FUNCTION_BLOCK FB_AxisControl EXTENDS FB_McAxis
VAR
  _eCheck                   : E_CHECK_STATE;  // pointer check

  _eAxisCycle,                                // cyclic AXIS_REF() and MC_Power check
  _eInit                    : E_PROGRESS;     // axis startup and init, get encoder type, get axis name

  _nAxisIndex               : UINT;           // know thyself
  _rTargetWindow            : LREAL := 0.1;   // TODO: get that from NC

  _stCtrl                   : POINTER TO ARRAY[1..PLC_CONSTANT.MAX_AXIS] OF ST_AXIS_CTRL;
  _stState                  : POINTER TO ARRAY[1..PLC_CONSTANT.MAX_AXIS] OF ST_AXIS_STATE;

  _Info                     : POINTER TO ARRAY[1..PLC_CONSTANT.MAX_AXIS] OF ST_AXIS_INFO;    // axis state and position data to read from
  _Data                     : POINTER TO ARRAY[1..PLC_CONSTANT.MAX_AXIS] OF ST_MOVE_DATA;    // structure for cyclic interface

  _NcParameter              : POINTER TO ARRAY[1..PLC_CONSTANT.MAX_AXIS] OF ST_NC_PARAMETER; // R/W struct for a single parameter
  _HomeParameter            : POINTER TO ARRAY[1..PLC_CONSTANT.MAX_AXIS] OF ST_HOMING;       // homing parameter for each axis

  _GearInParameter          : POINTER TO ARRAY[1..PLC_CONSTANT.MAX_AXIS] OF ST_GEAR_IN;
  _GearMultiMasterParameter : POINTER TO ARRAY[1..PLC_CONSTANT.MAX_AXIS] OF ST_GEAR_IN;

  _MotionOptions            : POINTER TO ARRAY[1..PLC_CONSTANT.MAX_AXIS] OF ST_MOTION_OPTIONS;


  _eCtrl,
  _eCtrlOld                 : E_AXIS_CTRL;

  _eCtrlParameterNr         : Tc2_MC2.MC_AxisParameter;

  _rParameterReadValue,
  _rParameterWrtValue       : LREAL;

  _eResult,
  _eResultOld               : E_PROGRESS;
  _eState                   : E_AXIS_STATE;

  // calibration options with limit switches and simulation
  _bCalibrationCam                : BOOL;

  _bLimitMin,
  _bLimitMax,
  _bCalibrationInput     AT %I*   : BOOL;
END_VAR

IF NOT Check() THEN RETURN; END_IF
//-----------------------------------------------------------------------------
// check _HomeParameter for calibration input options
//-----------------------------------------------------------------------------
_bCalibrationCam                    := GetCalibrationCam();
CalibrationCam                      := ADR(_bCalibrationCam);
//-----------------------------------------------------------------------------
//-----------------------------------------------------------------------------
Override                            := _Data^[_nAxisIndex].rOverride;


//-----------------------------------------------------------------------------
//-----------------------------------------------------------------------------
// cyclic call to MC_Power and AXIS_REF()
//-----------------------------------------------------------------------------
_eAxisCycle                         := Cycle();
//-----------------------------------------------------------------------------
//-----------------------------------------------------------------------------
// get command from outside world
//-----------------------------------------------------------------------------
_eCtrl                              := _stCtrl^[_nAxisIndex].eCtrl;

IF (_eCtrl <> _eCtrlOld)
THEN
  _eState                           := Cmd(_eCtrl);
  _eCtrlOld                         := _eCtrl;

  LogControl();

  _stState^[_nAxisIndex].eState     := _eState + TO_UINT(E_PROGRESS.BUSY);
END_IF
//-----------------------------------------------------------------------------
//-----------------------------------------------------------------------------
CASE _eState
OF
  E_AXIS_STATE.AXIS_INIT:
    //-------------------------------------------------------------------------
    // axis always requires one init from outside world at startup
    // _eInit has to be valid for other commands to be accepted in Cmd(_eCtrl)
    _eInit := _eResult              := AxisInit(TRUE);
    //-------------------------------------------------------------------------

  E_AXIS_STATE.AXIS_DISABLE:
    _eResult                        := AxisDisable(TRUE);

  E_AXIS_STATE.AXIS_ENABLE:
    _eResult                        := AxisEnable(TRUE);

  E_AXIS_STATE.AXIS_IDLE:
    _eResult                        := Idle(TRUE);

  E_AXIS_STATE.AXIS_HOME:
    _eResult                        := AxisHome(TRUE);

  E_AXIS_STATE.AXIS_MOVE_POS:
    _eResult                        := MovePosition(TRUE, _Data^[_nAxisIndex]);

  E_AXIS_STATE.AXIS_MOVE_VELO:
    _eResult                        := MoveVelocity(TRUE, _Data^[_nAxisIndex]);

  E_AXIS_STATE.AXIS_RESET:
    _eResult                        := AxisReset(TRUE);

  E_AXIS_STATE.AXIS_HALT:
    _eResult                        := AxisHalt(TRUE, _Data^[_nAxisIndex]);

  E_AXIS_STATE.AXIS_STOP:
    _eResult                        := AxisStop(TRUE, _Data^[_nAxisIndex]);

  E_AXIS_STATE.AXIS_MOVE_BUFFER:
    _eResult                        := MoveBufferPos(TRUE, _Data^[_nAxisIndex]);

  E_AXIS_STATE.AXIS_MOVE_BUFFER_VELO:
    _eResult                        := MoveBufferVelo(TRUE, _Data^[_nAxisIndex]);

  E_AXIS_STATE.AXIS_PARAMETER_READ:
    _eResult                        := ParameterRead(TRUE, _NcParameter^[_nAxisIndex].ParameterNumber);


  E_AXIS_STATE.AXIS_PARAMETER_WRITE:

  E_AXIS_STATE.AXIS_PARAMETER_WRITE_PERSISTENT:



  E_AXIS_STATE.AXIS_GEAR_IN:
  E_AXIS_STATE.AXIS_GEAR_OUT:
  E_AXIS_STATE.AXIS_GEAR_IN_MULTIMASTER:

ELSE
  _eResult                          := E_PROGRESS.ERROR;
END_CASE
//-----------------------------------------------------------------------------
// OnChange - log result and clear err nr on interface
//-----------------------------------------------------------------------------
IF (_eResult <> _eResultOld)
THEN
  LogResult();
  _Info^[_nAxisIndex].nErrorId     := 0;
  _eResultOld                      := _eResult;
END_IF
//-----------------------------------------------------------------------------
//-----------------------------------------------------------------------------
//  Output Data
//-----------------------------------------------------------------------------
//-----------------------------------------------------------------------------
CASE _eResult
OF
  E_PROGRESS.ERROR:
    _Info^[_nAxisIndex].bError      := TRUE;
    _Info^[_nAxisIndex].nErrorId    := ErrorId;
ELSE
    _Info^[_nAxisIndex].bError      := FALSE;
END_CASE
//-----------------------------------------------------------------------------
// state information is combined Info from Cmd(_eCtrl) and progress from method
//-----------------------------------------------------------------------------
_stState^[_nAxisIndex].eState       := _eState + TO_UINT(_eResult);
//-----------------------------------------------------------------------------
// Check ControlLoop
//-----------------------------------------------------------------------------
IF _AxisRef^.Status.ControlLoopClosed
THEN
  _Info^[_nAxisIndex].bEnabled      := TRUE;
ELSE
  _Info^[_nAxisIndex].bEnabled      := FALSE;
END_IF

_Info^[_nAxisIndex].bStandstill     := _AxisRef^.Status.NotMoving;

_Info^[_nAxisIndex].rActPos         := _AxisRef^.NcToPlc.ActPos;
_Info^[_nAxisIndex].rActVelo        := _AxisRef^.NcToPlc.ActVelo;
_Info^[_nAxisIndex].rPosDiff        := _AxisRef^.NcToPlc.PosDiff;

IF (_Info^[_nAxisIndex].rActPos < _Data^[_nAxisIndex].rSetPos + _rTargetWindow) AND
   (_Info^[_nAxisIndex].rActPos > _Data^[_nAxisIndex].rSetPos - _rTargetWindow) AND
    _Info^[_nAxisIndex].bStandstill
THEN
  _Info^[_nAxisIndex].bInTarget     := TRUE;
ELSE
  _Info^[_nAxisIndex].bInTarget     := FALSE;
END_IF
//-----------------------------------------------------------------------------
// copy CoupleState from axis
//-----------------------------------------------------------------------------
_Info^[_nAxisIndex].dwCoupleState   := _AxisRef^.NcToPlc.CoupleState;
//-----------------------------------------------------------------------------

PROPERTY AxisCtrl : pointer to ARRAY[1..PLC_CONSTANT.MAX_AXIS] OF st_axis_ctrl
SET
_stCtrl := AxisCtrl;
END_SET
END_PROPERTY

PROPERTY AxisData : pointer to ARRAY[1..PLC_CONSTANT.MAX_AXIS] OF st_move_data
SET
_Data := AxisData;
END_SET
END_PROPERTY

METHOD AxisDisable : E_PROGRESS
VAR_INPUT
  Execute           : BOOL;
END_VAR
VAR_INST
  _eState,
  _eResult          : E_PROGRESS;
  _rValue           : LREAL;
  _udiErr           : UDINT;
  _stMsg            : ST_Message;


END_VAR
IF NOT Check() THEN _eState := E_PROGRESS.ERROR; END_IF
IF NOT Execute THEN _eState := E_PROGRESS.INIT; END_IF

CASE _eState
OF
  E_PROGRESS.INIT:
    IF Execute 
    THEN
      memset(ADR(_stMsg),0,SIZEOF(_stMsg));
      _udiErr                       := 0;
      _rValue                       := 0;
      _eState                       := E_PROGRESS.BUSY;
    END_IF
END_CASE
CASE _eState
OF
  E_PROGRESS.BUSY:
    _eResult                        := Disable(FALSE);
    _eState                         := E_PROGRESS.WAITING;
END_CASE
CASE _eState
OF
  E_PROGRESS.WAITING:
    _eResult                        := Disable(TRUE);

    IF (_eResult = E_PROGRESS.DONE)
    THEN
      _eState                       := E_PROGRESS.WORKING;
    END_IF
END_CASE
CASE _eState
OF
  E_PROGRESS.WORKING:
    _eState                         := E_PROGRESS.DONE;
END_CASE

AxisDisable := _eState;
END_METHOD

METHOD AxisEnable : E_PROGRESS
VAR_INPUT
  Execute           : BOOL;
END_VAR
VAR_INST
  _eState,
  _eResult          : E_PROGRESS;
  _rValue           : LREAL;
  _udiErr           : UDINT;
  _stMsg            : ST_Message;


END_VAR
IF NOT Check() THEN _eState := E_PROGRESS.ERROR; END_IF
IF NOT Execute THEN _eState := E_PROGRESS.INIT; END_IF

CASE _eState
OF
  E_PROGRESS.INIT:
    IF Execute 
    THEN
      memset(ADR(_stMsg),0,SIZEOF(_stMsg));
      _udiErr                       := 0;
      _rValue                       := 0;
      _eState                       := E_PROGRESS.BUSY;
    END_IF
END_CASE
CASE _eState
OF
  E_PROGRESS.BUSY:
    _eResult                        := Enable(FALSE);
    _eState                         := E_PROGRESS.WAITING;
END_CASE
CASE _eState
OF
  E_PROGRESS.WAITING:
    _eResult                        := Enable(TRUE);

    IF (_eResult = E_PROGRESS.DONE)
    THEN
      _eState                       := E_PROGRESS.WORKING;
    END_IF
END_CASE
CASE _eState
OF
  E_PROGRESS.WORKING:
    _eState                         := E_PROGRESS.DONE;
END_CASE

AxisEnable := _eState;
END_METHOD

PROPERTY AxisGearInParameter : pointer to ARRAY[1..PLC_CONSTANT.MAX_AXIS] OF ST_GEAR_IN
SET
_GearInParameter := AxisGearInParameter;
END_SET
END_PROPERTY

METHOD AxisHalt : E_PROGRESS
VAR_INPUT
  Execute           : BOOL;
  Data              : ST_MOVE_DATA;
END_VAR
VAR_INST
  _eres,
  _eState           : E_PROGRESS;
  _rValue           : LREAL;
  _udiErr           : UDINT;
  _stMsg            : ST_Message;


END_VAR
IF NOT Check() THEN _eState := E_PROGRESS.ERROR; END_IF
IF NOT Execute THEN _eState := E_PROGRESS.INIT; END_IF

CASE _eState
OF
  E_PROGRESS.INIT:
    IF Execute 
    THEN
      memset(ADR(_stMsg),0,SIZEOF(_stMsg));
      _udiErr       := 0;
      _rValue       := 0;
      _eState       := E_PROGRESS.BUSY;
    END_IF
END_CASE
CASE _eState
OF
  E_PROGRESS.BUSY:
    _eState         := E_PROGRESS.WAITING;
    _eres           := Halt(
                            Execute := FALSE, 
                            Dec     := Data.rDec, 
                            Jerk    := Data.rJerk);
END_CASE
CASE _eState
OF
  E_PROGRESS.WAITING:
    _eres           := Halt(
                            Execute := TRUE, 
                            Dec     := Data.rDec, 
                            Jerk    := Data.rJerk);

    IF (_eres = E_PROGRESS.ERROR)
    THEN
        _eState     := E_PROGRESS.ERROR;
    ELSIF (_eres = E_PROGRESS.DONE)
    THEN 
      _eState       := E_PROGRESS.WORKING;
    END_IF
END_CASE
CASE _eState
OF
  E_PROGRESS.WORKING:
    _eState         := E_PROGRESS.DONE;
    _eres           := Halt(
                            Execute := FALSE, 
                            Dec     := Data.rDec, 
                            Jerk    := Data.rJerk);
END_CASE

AxisHalt := _eState;
END_METHOD

METHOD AxisHome : E_PROGRESS
VAR_INPUT
  Execute           : BOOL;
END_VAR
VAR_INST
  _eres,
  _eState           : E_PROGRESS;
  _rValue           : LREAL;
  _udiErr           : UDINT;
  _stMsg            : ST_Message;


END_VAR
IF NOT Check() THEN _eState := E_PROGRESS.ERROR; END_IF
IF NOT Execute THEN _eState := E_PROGRESS.INIT; END_IF

CASE _eState
OF
  E_PROGRESS.INIT:
    IF Execute 
    THEN
      memset(ADR(_stMsg),0,SIZEOF(_stMsg));
      _udiErr               := 0;
      _rValue               := 0;

      IF (_AxisRef^.Status.Homed)
      THEN
        _eState             := E_PROGRESS.BUSY;
      ELSE
        _eState             := E_PROGRESS.PREPARE;
      END_IF
    END_IF
END_CASE
CASE _eState
OF
  E_PROGRESS.BUSY:
    _eState                 := E_PROGRESS.STARTUP;
    _eres                   := Home(Execute   := FALSE,
                                    Position  := _HomeParameter^[_nAxisIndex].stHomingParam.Position,
                                    HomingMode:= Tc2_MC2.MC_HomingMode.MC_ResetCalibration,
                                    Options   := _HomeParameter^[_nAxisIndex].stHomingParam.Options);

END_CASE
CASE _eState
OF
  E_PROGRESS.STARTUP:
    _Info^[_nAxisIndex].bReferenced   := FALSE;

    _eres                   := Home(
                                    Execute   := TRUE,
                                    Position  := _HomeParameter^[_nAxisIndex].stHomingParam.Position,
                                    HomingMode:= Tc2_MC2.MC_HomingMode.MC_ResetCalibration,
                                    Options   := _HomeParameter^[_nAxisIndex].stHomingParam.Options);
    IF (_eres = E_PROGRESS.DONE)
    THEN
      _eState               := E_PROGRESS.PREPARE;
    END_IF
END_CASE
CASE _eState
OF
  E_PROGRESS.PREPARE:
      _eState               := E_PROGRESS.READY;

      _eres                 := Home(
                                    Execute   := FALSE,
                                    Position  := _HomeParameter^[_nAxisIndex].stHomingParam.Position,
                                    HomingMode:= Tc2_MC2.MC_HomingMode.MC_ResetCalibration,
                                    Options   := _HomeParameter^[_nAxisIndex].stHomingParam.Options);
END_CASE
CASE _eState
OF
  E_PROGRESS.READY:
    _eState                 := E_PROGRESS.WAITING;

END_CASE
CASE _eState
OF
  E_PROGRESS.WAITING:
    _eres                   := Home(
                                    Execute   := TRUE,
                                    Position  := _HomeParameter^[_nAxisIndex].stHomingParam.Position,
                                    HomingMode:= _HomeParameter^[_nAxisIndex].stHomingParam.HomingMode,
                                    Options   := _HomeParameter^[_nAxisIndex].stHomingParam.Options);

    IF (_eres = E_PROGRESS.ERROR)
    THEN
      _eState               := E_PROGRESS.ERROR;
    ELSIF (_eres = E_PROGRESS.DONE)
    THEN
      _eState               := E_PROGRESS.WORKING;
    END_IF
END_CASE
CASE _eState
OF
  E_PROGRESS.WORKING:
    _eState                 := E_PROGRESS.DONE;

    _eres                   := Home(
                                    Execute   := FALSE,
                                    Position  := _HomeParameter^[_nAxisIndex].stHomingParam.Position,
                                    HomingMode:= _HomeParameter^[_nAxisIndex].stHomingParam.HomingMode,
                                    Options   := _HomeParameter^[_nAxisIndex].stHomingParam.Options);
END_CASE

AxisHome := _eState;
END_METHOD

PROPERTY AxisIndex : uint
SET
END_SET
END_PROPERTY

PROPERTY AxisInfo : pointer to ARRAY[1..PLC_CONSTANT.MAX_AXIS] OF ST_AXIS_INFO
SET
_Info := AxisInfo;
END_SET
END_PROPERTY

METHOD PRIVATE AxisInit : E_PROGRESS
VAR_INPUT
  Execute           : BOOL;
END_VAR
VAR_INST
  _eResult,
  _eState           : E_PROGRESS;
  _rValue           : LREAL;
  _stMsg            : ST_Message;

  // access to CoE register
  _sDeviceName      : STRING(256) := 'NO NAME';
  _fbCoeRead				: Tc2_MC2_Drive.FB_CoERead;
END_VAR
IF NOT Check() THEN _eState := E_PROGRESS.ERROR; END_IF
IF NOT Execute THEN _eState := E_PROGRESS.INIT; END_IF

CASE _eState
OF
  E_PROGRESS.INIT:
    IF Execute 
    THEN
      memset(ADR(_stMsg),0,SIZEOF(_stMsg));

      _nErrorId                     := 0;
      _rValue                       := 0;
      _eState                       := E_PROGRESS.BUSY;
      _eInit                        := _eState;
    END_IF
END_CASE
CASE _eState
OF
  E_PROGRESS.BUSY:
    _eState                         := E_PROGRESS.STARTUP;
    _eResult                        := StartUp(FALSE);
END_CASE
CASE _eState
OF
  E_PROGRESS.STARTUP:
    _eResult                        := StartUp(TRUE);
    IF (_eResult = E_PROGRESS.DONE)
    THEN
      _eState                       := E_PROGRESS.PREPARE;
      _eResult                      := AxisReset(FALSE);
    ELSIF (_eResult = E_PROGRESS.ERROR)
    THEN
      _eState                       := _eResult;

      _stMsg.eType                  := E_MessageType.eMessageError;
      _stMsg.eDevice                := e_Device.Axis + TO_DINT(_AxisRef^.NcToPlc.AxisId);
      _stMsg.eSubdevice             := e_Subdevice.fbAxis_StartUp;
      _stMsg.iErrorNumber := _nErrorId  := 6666;

      _stMsg.sText                  := TO_STRING(_eState);
      f_MessageSet(_stMsg);

    END_IF
END_CASE
CASE _eState
OF
  E_PROGRESS.PREPARE:
    _eResult                        := AxisReset(TRUE);
    IF (_eResult = E_PROGRESS.DONE)
    THEN
      _fbCoeRead(
                Execute               := FALSE,
                NetId                 := _AxisRef^.ADS.NetId, 
                Axis                  := _AxisRef^);
  
      IF (EncoderType <> 1)
      THEN
        memset(ADR(_sDeviceName),0,SIZEOF(_sDeviceName));
  
        _eState                       := E_PROGRESS.READY;
      ELSE
        _eState                       := E_PROGRESS.WORKING;
      END_IF
    ELSIF (_eResult = E_PROGRESS.ERROR)
    THEN
      _eState                       := _eResult;

      _stMsg.eType                  := E_MessageType.eMessageError;
      _stMsg.eDevice                := e_Device.Axis + TO_DINT(_AxisRef^.NcToPlc.AxisId);
      _stMsg.eSubdevice             := e_Subdevice.fbAxis_StartupReset;
      _stMsg.iErrorNumber           := ErrorId;

      _stMsg.sText                  := TO_STRING(_eState);
      f_MessageSet(_stMsg);

    END_IF
END_CASE
CASE _eState
OF
  E_PROGRESS.READY:
    _eResult                        := Reset(FALSE);
    // get manufacturer device name in CoE
    _fbCoeRead.Index                := 16#1008;
    _fbCoeRead.SubIndex             := 0;
    _fbCoeRead.pDstBuf              := ADR(_sDeviceName);
    _fbCoeRead.BufLen               := SIZEOF(_sDeviceName);

    _fbCoeRead(
              Execute               := TRUE,
              NetId                 := _AxisRef^.ADS.NetId, 
              Axis                  := _AxisRef^);

    IF _fbCoeRead.Busy
    THEN
      _eState                       := E_PROGRESS.WAITING;
    END_IF
END_CASE
CASE _eState
OF
  E_PROGRESS.WAITING:
    _fbCoeRead(
              NetId                 := _AxisRef^.ADS.NetId, 
              Axis                  := _AxisRef^);

    IF (_fbCoeRead.Error)
    THEN
      _eState                       := E_PROGRESS.ERROR;
      _Info^[_nAxisIndex].nErrorId := SEL((_fbCoeRead.CANopenErrId > 0), _fbCoeRead.AdsErrId, _fbCoeRead.CANopenErrId);

      _fbCoeRead(
                Execute             := FALSE,
                NetId               := _AxisRef^.ADS.NetId, 
                Axis                := _AxisRef^);

      _stMsg.eType                  := E_MessageType.eMessageError;
      _stMsg.eDevice                := e_Device.Axis + TO_DINT(_AxisRef^.NcToPlc.AxisId);
      _stMsg.eSubdevice             := e_Subdevice.fbCoeRead;

      _stMsg.iErrorNumber           := SEL((_fbCoeRead.CANopenErrId > 0), _fbCoeRead.AdsErrId, _fbCoeRead.CANopenErrId);

      _stMsg.sText                  := TO_STRING(_eState);
      f_MessageSet(_stMsg);

    ELSIF NOT _fbCoeRead.Busy
    THEN
      _eState                       := E_PROGRESS.WORKING;
    END_IF
END_CASE
CASE _eState
OF
  E_PROGRESS.WORKING:
    _eState                         := E_PROGRESS.DONE;

    // set default for axis release
    AxisEnableNegative              := TRUE;
    AxisEnablePositive              := TRUE;

    // clear fb
    _fbCoeRead(
              Execute               := FALSE,
              NetId                 := _AxisRef^.ADS.NetId, 
              Axis                  := _AxisRef^);

    _stMsg.eType                    := E_MessageType.eMessageInfo;
    _stMsg.eDevice                  := e_Device.Axis + TO_DINT(_AxisRef^.NcToPlc.AxisId);
    _stMsg.eSubdevice               := e_Subdevice.fbAxis_StartUp;
    _stMsg.iErrorNumber             := 0;
    _stMsg.sText                    := TO_STRING(_eState);
    f_MessageSet(_stMsg);
END_CASE

AxisInit := _eState;
END_METHOD

PROPERTY AxisNcParameter : pointer to ARRAY[1..PLC_CONSTANT.MAX_AXIS] OF st_nc_parameter
SET
_NcParameter := AxisNcParameter;
END_SET
END_PROPERTY

PROPERTY AxisNcParameterValue : Lreal
GET
AxisNcParameterValue := _rParameterReadValue;
END_GET
END_PROPERTY

METHOD AxisReset : E_PROGRESS
VAR_INPUT
  Execute           : BOOL;
END_VAR
VAR_INST
  _eres,
  _eState           : E_PROGRESS;
  _rValue           : LREAL;
  _udiErr           : UDINT;
  _stMsg            : ST_Message;


END_VAR
IF NOT Check() THEN _eState := E_PROGRESS.ERROR; END_IF
IF NOT Execute THEN _eState := E_PROGRESS.INIT; END_IF

CASE _eState
OF
  E_PROGRESS.INIT:
    IF Execute 
    THEN
      memset(ADR(_stMsg),0,SIZEOF(_stMsg));
      _udiErr                       := 0;
      _rValue                       := 0;
      _eState                       := E_PROGRESS.BUSY;
    END_IF
END_CASE
CASE _eState
OF
  E_PROGRESS.BUSY:
    _eres                           := Reset(FALSE);
    _eState                         := E_PROGRESS.WAITING;
END_CASE
CASE _eState
OF
  E_PROGRESS.WAITING:

    _eres                           := Reset(TRUE);
    IF (_eres = E_PROGRESS.DONE)
    THEN
      _eState                       := E_PROGRESS.WORKING;
    ELSIF (_eres = E_PROGRESS.ERROR)
    THEN
      _eState                       := E_PROGRESS.ERROR;
    END_IF
END_CASE
CASE _eState
OF
  E_PROGRESS.WORKING:
    _eres                           := Reset(FALSE);
    _eState                         := E_PROGRESS.DONE;
END_CASE

AxisReset := _eState;
END_METHOD

PROPERTY AxisState : pointer to ARRAY[1..PLC_CONSTANT.MAX_AXIS] OF ST_AXIS_STATE
SET
_stState := AxisState;
END_SET
END_PROPERTY

METHOD AxisStop : E_PROGRESS
VAR_INPUT
  Execute           : BOOL;
  Data              : ST_MOVE_DATA;
END_VAR
VAR_INST
  _eres,
  _eState           : E_PROGRESS;
  _rValue           : LREAL;
  _udiErr           : UDINT;
  _stMsg            : ST_Message;


END_VAR
IF NOT Check() THEN _eState := E_PROGRESS.ERROR; END_IF
IF NOT Execute THEN _eState := E_PROGRESS.INIT; END_IF

CASE _eState
OF
  E_PROGRESS.INIT:
    IF Execute 
    THEN
      memset(ADR(_stMsg),0,SIZEOF(_stMsg));
      _udiErr       := 0;
      _rValue       := 0;
      _eState       := E_PROGRESS.BUSY;
    END_IF
END_CASE
CASE _eState
OF
  E_PROGRESS.BUSY:
    _eState         := E_PROGRESS.WAITING;
    _eres           := Stop(
                            Execute := FALSE, 
                            Dec     := Data.rDec, 
                            Jerk    := Data.rJerk);
END_CASE
CASE _eState
OF
  E_PROGRESS.WAITING:
    _eres           := Stop(
                            Execute := TRUE, 
                            Dec     := Data.rDec, 
                            Jerk    := Data.rJerk);

    IF (_eres = E_PROGRESS.ERROR)
    THEN
        _eState     := E_PROGRESS.ERROR;
    ELSIF (_eres = E_PROGRESS.DONE)
    THEN 
      _eState       := E_PROGRESS.WORKING;
    END_IF
END_CASE
CASE _eState
OF
  E_PROGRESS.WORKING:
    _eState         := E_PROGRESS.DONE;
    _eres           := Stop(
                            Execute := FALSE, 
                            Dec     := Data.rDec, 
                            Jerk    := Data.rJerk);
END_CASE

AxisStop := _eState;
END_METHOD

METHOD PRIVATE Check : BOOL

IF (_nAxisIndex < 1) OR
   (_nAxisIndex > PLC_CONSTANT.MAX_AXIS)
THEN
  _eCheck                 := E_CHECK_STATE.AXIS_INDEX_OUT_OF_RANGE;
  RETURN;
END_IF

IF NOT (_AxisRef <> 0)
THEN
  _eCheck                 := E_CHECK_STATE.AXIS_REF_POINTER_INVALID;
  RETURN;
END_IF

IF NOT (_stCtrl <> 0)
THEN
  _eCheck                 := E_CHECK_STATE.AXIS_CTRL_POINTER_INVALID;
  RETURN;
END_IF

IF NOT (_stState <> 0)
THEN
  _eCheck                 := E_CHECK_STATE.AXIS_STATE_POINTER_INVALID;
  RETURN;
END_IF

IF NOT (_Info <> 0)
THEN
  _eCheck                 := E_CHECK_STATE.AXIS_INFO_POINTER_INVALID;
  RETURN;
END_IF

IF NOT (_Data <> 0)
THEN
  _eCheck                 := E_CHECK_STATE.AXIS_DATA_POINTER_INVALID;
  RETURN;
END_IF

IF NOT (_NcParameter <> 0)
THEN
  _eCheck                 := E_CHECK_STATE.AXIS_NC_PARAMETER_POINTER_INVALID;
  RETURN;
END_IF

IF NOT (_HomeParameter <> 0)
THEN
  _eCheck                 := E_CHECK_STATE.AXIS_HOME_PARAMETER_POINTER_INVALID;
  RETURN;
END_IF

IF NOT (_GearInParameter <> 0)
THEN
  _eCheck                 := E_CHECK_STATE.AXIS_GEAR_IN_PARAMETER_POINTER_INVALID;
  RETURN;
END_IF
  
IF NOT (_GearMultiMasterParameter <> 0)
THEN
  _eCheck                 := E_CHECK_STATE.AXIS_GEAR_IN_MULTIMASTER_POINTER_INVALID;
  RETURN;
END_IF

IF NOT (_MotionOptions <> 0)
THEN
  _eCheck                 := E_CHECK_STATE.AXIS_MOTION_OPTIONS_POINTER_INVALID;
  RETURN;
END_IF

(*
-------------------------------------------------------------------------------
	NaN INF check
-------------------------------------------------------------------------------
*)
IF NOT IsFinite(F_LReal(_Data^[_nAxisIndex].rSetPos))
THEN
	_Data^[_nAxisIndex].rSetPos := 0.0;
END_IF

IF NOT IsFinite(F_LReal(_Data^[_nAxisIndex].rSetVelo))
THEN
	_Data^[_nAxisIndex].rSetVelo := 0.0;
END_IF

IF NOT IsFinite(F_LReal(_Data^[_nAxisIndex].rAcc))
THEN
	_Data^[_nAxisIndex].rAcc := 0.0;
END_IF

IF NOT IsFinite(F_LReal(_Data^[_nAxisIndex].rDec))
THEN
	_Data^[_nAxisIndex].rDec := 0.0;
END_IF

IF NOT IsFinite(F_LReal(_Data^[_nAxisIndex].rOverride))
THEN
	_Data^[_nAxisIndex].rOverride := 0.0;
END_IF


_eCheck                   := E_CHECK_STATE.CHECK_DONE;
Check                     := TRUE;
END_METHOD

METHOD Cmd : E_AXIS_STATE
VAR_INPUT
  eCmd      : E_AXIS_CTRL;
END_VAR
VAR_INST
  _estate   : E_AXIS_STATE;
  _eres     : E_PROGRESS;
END_VAR

CASE eCmd
OF
  E_AXIS_CTRL.AXIS_INIT:
    _eInit                  := AxisInit(FALSE);
    _estate                 := E_AXIS_STATE.AXIS_INIT;
ELSE
  IF (_eInit <> E_PROGRESS.DONE)
  THEN
    _estate                 := E_AXIS_STATE.AXIS_INVALID;
  ELSE
    CASE eCmd
    OF
      E_AXIS_CTRL.AXIS_DISABLE:
        _eres               := AxisDisable(FALSE);
        _estate             := E_AXIS_STATE.AXIS_DISABLE;
    
      E_AXIS_CTRL.AXIS_ENABLE:
        _eres               := AxisEnable(FALSE);
        _estate             := E_AXIS_STATE.AXIS_ENABLE;
    
      E_AXIS_CTRL.AXIS_IDLE:
        _eres               := Idle(FALSE);
        _estate             := E_AXIS_STATE.AXIS_IDLE;
    
      E_AXIS_CTRL.AXIS_HOME:
        _eres               := AxisHome(FALSE);
        _estate             := E_AXIS_STATE.AXIS_HOME;
    
      E_AXIS_CTRL.AXIS_MOVE_POS:
        _eres               := MovePosition(FALSE, _Data^[_nAxisIndex]);
        _estate             := E_AXIS_STATE.AXIS_MOVE_POS;
    
      E_AXIS_CTRL.AXIS_MOVE_VELO:
        _eres               := MoveVelocity(FALSE, _Data^[_nAxisIndex]);
        _estate             := E_AXIS_STATE.AXIS_MOVE_VELO;
    
      E_AXIS_CTRL.AXIS_RESET:
        _eres               := AxisReset(FALSE);
        _estate             := E_AXIS_STATE.AXIS_RESET;
    
      E_AXIS_CTRL.AXIS_HALT:
        _eres               := AxisHalt(FALSE, _Data^[_nAxisIndex]);
        _estate             := E_AXIS_STATE.AXIS_HALT;
    
      E_AXIS_CTRL.AXIS_STOP:
        _eres               := AxisStop(FALSE, _Data^[_nAxisIndex]);
        _estate             := E_AXIS_STATE.AXIS_STOP;
    
      E_AXIS_CTRL.AXIS_MOVE_BUFFER:
        _eres               := MoveBufferPos(FALSE, _Data^[_nAxisIndex]);
        _estate             := E_AXIS_STATE.AXIS_MOVE_BUFFER;
    
      E_AXIS_CTRL.AXIS_MOVE_BUFFER_VELO:
        _eres               := MoveBufferVelo(FALSE, _Data^[_nAxisIndex]);
        _estate             := E_AXIS_STATE.AXIS_MOVE_BUFFER_VELO;
    
      E_AXIS_CTRL.AXIS_PARAMETER_READ:
        _eCtrlParameterNr   := _NcParameter^[_nAxisIndex].ParameterNumber;
        _eres               := ParameterRead(FALSE, _eCtrlParameterNr);
        _estate             := E_AXIS_STATE.AXIS_PARAMETER_READ;

      E_AXIS_CTRL.AXIS_PARAMETER_WRITE:
        _eCtrlParameterNr   := _NcParameter^[_nAxisIndex].ParameterNumber;
        _rParameterWrtValue := _NcParameter^[_nAxisIndex].rValue;

        _estate             := E_AXIS_STATE.AXIS_PARAMETER_WRITE;

      E_AXIS_CTRL.AXIS_PARAMETER_WRITE_PERSISTENT:
        _eCtrlParameterNr   := _NcParameter^[_nAxisIndex].ParameterNumber;
        _rParameterWrtValue := _NcParameter^[_nAxisIndex].rValue;

        _estate             := E_AXIS_STATE.AXIS_PARAMETER_WRITE_PERSISTENT;
    
      E_AXIS_CTRL.AXIS_GEAR_IN:
        _estate             := E_AXIS_STATE.AXIS_GEAR_IN;
    
      E_AXIS_CTRL.AXIS_GEAR_OUT:
        _estate             := E_AXIS_STATE.AXIS_GEAR_OUT;
    
      E_AXIS_CTRL.AXIS_GEAR_IN_MULTIMASTER:
        _estate             := E_AXIS_STATE.AXIS_GEAR_IN_MULTIMASTER;
    ELSE
      _estate               := E_AXIS_STATE.AXIS_INVALID;
      _eres                 := E_PROGRESS.ERROR; // wrong note! wrong note!
    END_CASE
  END_IF // _eInit
END_CASE

Cmd                         := _estate;
END_METHOD

METHOD PRIVATE GetCalibrationCam : BOOL
VAR_INST
  _bCal     : Bool;
END_VAR
IF _HomeParameter^[_nAxisIndex].stHomingParam.SimulateHomeSensor
THEN
	IF (_AxisRef^.NcToPlc.HomingState < 4)
  THEN
		_bCal := TRUE;
	ELSE
		_bCal := FALSE;
	END_IF
ELSIF _HomeParameter^[_nAxisIndex].stHomingParam.HomeOnLimitMin
THEN
	_bCal := _bLimitMin XOR _HomeParameter^[_nAxisIndex].stHomingParam.InvertHomeSensor;

ELSIF _HomeParameter^[_nAxisIndex].stHomingParam.HomeOnLimitMax
THEN
	_bCal := _bLimitMax XOR _HomeParameter^[_nAxisIndex].stHomingParam.InvertHomeSensor;
ELSE
	_bCal := _bCalibrationInput XOR _HomeParameter^[_nAxisIndex].stHomingParam.InvertHomeSensor;
END_IF

GetCalibrationCam := _bCal;
END_METHOD

PROPERTY HomingParameter : pointer to ARRAY[1..PLC_CONSTANT.MAX_AXIS] OF st_homing
SET
_HomeParameter := HomingParameter;
END_SET
END_PROPERTY

METHOD Idle : E_PROGRESS
VAR_INPUT
  Execute           : BOOL;
END_VAR
VAR_INST
  _eResult,
  _eState           : E_PROGRESS;
  _rValue           : LREAL;
  _udiErr           : UDINT;
  _stMsg            : ST_Message;


END_VAR
IF NOT Check() THEN _eState := E_PROGRESS.ERROR; END_IF
IF NOT Execute THEN _eState := E_PROGRESS.INIT; END_IF

CASE _eState
OF
  E_PROGRESS.INIT:
    IF Execute 
    THEN
      memset(ADR(_stMsg),0,SIZEOF(_stMsg));
      _udiErr                       := 0;
      _rValue                       := 0;
      _eState                       := E_PROGRESS.BUSY;
    END_IF
END_CASE
CASE _eState
OF
  E_PROGRESS.BUSY:
    IF _AxisRef^.Status.Error
    THEN
      _eResult                      := Reset(FALSE);
      _eState                       := E_PROGRESS.STARTUP;
    ELSE
      _eState                       := E_PROGRESS.PREPARE;
    END_IF
END_CASE
CASE _eState
OF
  E_PROGRESS.STARTUP:
    _eResult                        := Reset(TRUE);

    IF (_eResult = E_PROGRESS.DONE)
    THEN
      _eState                       := E_PROGRESS.PREPARE;
    END_IF
END_CASE
CASE _eState
OF
  E_PROGRESS.PREPARE:
    _eResult                        := Reset(FALSE);
    _eResult                        := Enable(FALSE);
    _eState                         := E_PROGRESS.READY;
END_CASE
CASE _eState
OF
  E_PROGRESS.READY:
    _eResult                        := Enable(TRUE);

    IF (_eResult = E_PROGRESS.DONE)
    THEN
      _eState                       := E_PROGRESS.WAITING;

    ELSIF (_eResult = E_PROGRESS.ERROR)
    THEN
      _eState                       := E_PROGRESS.BUSY;
    END_IF
END_CASE
CASE _eState
OF
  E_PROGRESS.WAITING:
    Enable(FALSE);
    _eState                         := E_PROGRESS.WORKING;
END_CASE
CASE _eState
OF
  E_PROGRESS.WORKING:
    _eState                         := E_PROGRESS.DONE;
END_CASE

Idle := _eState;
END_METHOD

METHOD PRIVATE LogControl
VAR_INST
  _sResult,
  _sCtrl            : STRING(30);

  _stMsg            : ST_Message;
END_VAR

  _stMsg.eType               := E_MessageType.eMessageInfo;
  _stMsg.eDevice             := E_Device.Axis + TO_DINT(_AxisRef^.NcToPlc.AxisId);
  _stMsg.eSubdevice          := e_Subdevice.AxisMode;
  _stMsg.iErrorNumber        := _AxisRef^.NcToPlc.AxisId;

  _sCtrl                     := concat('E_AXIS_CTRL', '.');
  _sCtrl                     := concat(_sCtrl, TO_STRING(_eCtrl));

  _stMsg.sText               := concat('new command: ', _sResult);
  f_MessageSet(_stMsg);
END_METHOD

METHOD PRIVATE LogResult
VAR_INST
  _sResult,
  _sCtrl            : STRING(30);

  _stMsg            : ST_Message;
END_VAR

  _stMsg.eType               := E_MessageType.eMessageInfo;
  _stMsg.eDevice             := E_Device.Axis + TO_DINT(_AxisRef^.NcToPlc.AxisId);
  _stMsg.eSubdevice          := e_Subdevice.AxisMode;
  _stMsg.iErrorNumber        := _AxisRef^.NcToPlc.AxisId;

  _sCtrl                     := concat('E_AXIS_CTRL', '.');
  _sCtrl                     := concat(_sCtrl, TO_STRING(_eCtrl));

  _sResult                   := concat('E_PROGRESS', '.');
  _sResult                   := concat(_sResult, TO_STRING(_eResult));

  _stMsg.sText               := concat(_sCtrl, ' ');
  _stMsg.sText               := concat(_sCtrl, _sResult);
  f_MessageSet(_stMsg);
END_METHOD

PROPERTY MotionOptions : pointer to ARRAY[1..PLC_CONSTANT.MAX_AXIS] OF ST_MOTION_OPTIONS
SET
_MotionOptions := MotionOptions;
END_SET
END_PROPERTY

METHOD MoveBufferPos : E_PROGRESS
VAR_INPUT
  Enable            : BOOL;
  Data              : ST_MOVE_DATA;
END_VAR
VAR_INST
  _BufferMode       : Tc2_MC2.MC_BufferMode;
  _eres,
  _eState           : E_PROGRESS;
  _rValue           : LREAL;
  _udiErr           : UDINT;
  _stMsg            : ST_Message;
END_VAR
IF NOT Check() THEN _eState := E_PROGRESS.ERROR; END_IF
IF NOT Enable THEN _eState := E_PROGRESS.INIT; END_IF

CASE _eState
OF
  E_PROGRESS.INIT:
    IF Enable 
    THEN
      memset(ADR(_stMsg),0,SIZEOF(_stMsg));
      _udiErr       := 0;
      _rValue       := 0;
      _eState       := E_PROGRESS.BUSY;
    END_IF
END_CASE
CASE _eState
OF
  E_PROGRESS.BUSY:
    _eState         := E_PROGRESS.WORKING;
    _BufferMode     := _MotionOptions^[_nAxisIndex].eBufferMode;
    _eres           := MovePosBuffer(
                                  Enable      := FALSE, 
                                  Position    := Data.rSetPos, 
                                  Vel         := Data.rSetVelo, 
                                  Acc         := Data.rAcc, 
                                  Dec         := Data.rDec, 
                                  Jerk        := Data.rJerk, 
                                  BufferMode  := _BufferMode);

END_CASE
CASE _eState
OF
  E_PROGRESS.WORKING:
    _BufferMode     := _MotionOptions^[_nAxisIndex].eBufferMode;
    _eres           := MovePosBuffer(
                                  Enable      := TRUE, 
                                  Position    := Data.rSetPos, 
                                  Vel         := Data.rSetVelo, 
                                  Acc         := Data.rAcc, 
                                  Dec         := Data.rDec, 
                                  Jerk        := Data.rJerk, 
                                  BufferMode  := _BufferMode);
    IF (_eres = E_PROGRESS.ERROR)
    THEN
      _eState := E_PROGRESS.ERROR;
    END_IF
END_CASE

MoveBufferPos := _eState;
END_METHOD

METHOD MoveBufferVelo : E_PROGRESS
VAR_INPUT
  Enable            : BOOL;
  Data              : ST_MOVE_DATA;
END_VAR
VAR_INST
  _BufferMode       : Tc2_MC2.MC_BufferMode;
  _eres,
  _eState           : E_PROGRESS;
  _rValue           : LREAL;
  _udiErr           : UDINT;
  _stMsg            : ST_Message;
END_VAR
IF NOT Check() THEN _eState := E_PROGRESS.ERROR; END_IF
IF NOT Enable THEN _eState := E_PROGRESS.INIT; END_IF

CASE _eState
OF
  E_PROGRESS.INIT:
    IF Enable 
    THEN
      memset(ADR(_stMsg),0,SIZEOF(_stMsg));
      _udiErr       := 0;
      _rValue       := 0;
      _eState       := E_PROGRESS.BUSY;
    END_IF
END_CASE
CASE _eState
OF
  E_PROGRESS.BUSY:
    _eState         := E_PROGRESS.WORKING;
    _BufferMode     := _MotionOptions^[_nAxisIndex].eBufferMode;
    _eres           := MoveVeloBuffer(
                                  Enable      := FALSE, 
                                  Velocity    := Data.rSetVelo, 
                                  Acc         := Data.rAcc, 
                                  Dec         := Data.rDec, 
                                  Jerk        := Data.rJerk, 
                                  BufferMode  := _BufferMode);

END_CASE
CASE _eState
OF
  E_PROGRESS.WORKING:
    _BufferMode     := _MotionOptions^[_nAxisIndex].eBufferMode;
    _eres           := MoveVeloBuffer(
                                  Enable      := TRUE, 
                                  Velocity    := Data.rSetVelo, 
                                  Acc         := Data.rAcc, 
                                  Dec         := Data.rDec, 
                                  Jerk        := Data.rJerk, 
                                  BufferMode  := _BufferMode);
    IF (_eres = E_PROGRESS.ERROR)
    THEN
      _eState := E_PROGRESS.ERROR;
    END_IF
END_CASE

MoveBufferVelo := _eState;
END_METHOD

METHOD MovePosition : E_PROGRESS
VAR_INPUT
  Execute           : BOOL;
  Data              : ST_MOVE_DATA;
END_VAR
VAR_INST
  _eres,
  _eState           : E_PROGRESS;
  _rValue           : LREAL;
  _udiErr           : UDINT;
  _stMsg            : ST_Message;


END_VAR
IF NOT Check() THEN _eState := E_PROGRESS.ERROR; END_IF
IF NOT Execute THEN _eState := E_PROGRESS.INIT; END_IF

CASE _eState
OF
  E_PROGRESS.INIT:
    IF Execute 
    THEN
      memset(ADR(_stMsg),0,SIZEOF(_stMsg));
      _udiErr               := 0;
      _rValue               := 0;
      _eState               := E_PROGRESS.BUSY;
    END_IF
END_CASE
CASE _eState
OF
  E_PROGRESS.BUSY:
    _eState                 := E_PROGRESS.WAITING;
    _eres                   := MoveToPos(
                                      Execute    := FALSE, 
                                      Position   := Data.rSetPos, 
                                      Vel        := Data.rSetVelo, 
                                      Acc        := Data.rAcc, 
                                      Dec        := Data.rDec, 
                                      Jerk       := Data.rJerk, 
                                      BufferMode := Tc2_MC2.MC_BufferMode.MC_Aborting);
END_CASE
CASE _eState
OF
  E_PROGRESS.WAITING:
    _eres                   := MoveToPos(
                                      Execute    := TRUE, 
                                      Position   := Data.rSetPos, 
                                      Vel        := Data.rSetVelo, 
                                      Acc        := Data.rAcc, 
                                      Dec        := Data.rDec, 
                                      Jerk       := Data.rJerk, 
                                      BufferMode := Tc2_MC2.MC_BufferMode.MC_Aborting);

    IF (_eres = E_PROGRESS.ERROR)
    THEN
        _eState             := E_PROGRESS.ERROR;
    ELSIF (_eres = E_PROGRESS.DONE)
    THEN 
      _eState               := E_PROGRESS.WORKING;
    END_IF
END_CASE
CASE _eState
OF
  E_PROGRESS.WORKING:
    _eState                 := E_PROGRESS.DONE;
    _eres                   := MoveToPos(
                                      Execute    := FALSE, 
                                      Position   := Data.rSetPos, 
                                      Vel        := Data.rSetVelo, 
                                      Acc        := Data.rAcc, 
                                      Dec        := Data.rDec, 
                                      Jerk       := Data.rJerk, 
                                      BufferMode := Tc2_MC2.MC_BufferMode.MC_Aborting);
END_CASE

MovePosition := _eState;
END_METHOD

METHOD MoveVelocity : E_PROGRESS
VAR_INPUT
  Execute           : BOOL;
  Data              : ST_MOVE_DATA;
END_VAR
VAR_INST
  _eres,
  _eState           : E_PROGRESS;
  _rValue           : LREAL;
  _udiErr           : UDINT;
  _stMsg            : ST_Message;
END_VAR
IF NOT Check() THEN _eState := E_PROGRESS.ERROR; END_IF
IF NOT Execute THEN _eState := E_PROGRESS.INIT; END_IF

CASE _eState
OF
  E_PROGRESS.INIT:
    IF Execute 
    THEN
      memset(ADR(_stMsg),0,SIZEOF(_stMsg));
      _udiErr               := 0;
      _rValue               := 0;
      _eState               := E_PROGRESS.BUSY;
    END_IF
END_CASE
CASE _eState
OF
  E_PROGRESS.BUSY:
    _eState                 := E_PROGRESS.WAITING;
    _eres                   := MoveVelo(
                                    Execute     := FALSE, 
                                    Velocity    := Data.rSetVelo, 
                                    Acc         := Data.rAcc, 
                                    Dec         := Data.rDec, 
                                    Jerk        := Data.rJerk, 
                                    Direction   := Data.iDirection, 
                                    BufferMode  := Tc2_MC2.MC_BufferMode.MC_Aborting);
END_CASE
CASE _eState
OF
  E_PROGRESS.WAITING:
    _eres                   := MoveVelo(
                                    Execute     := TRUE, 
                                    Velocity    := Data.rSetVelo, 
                                    Acc         := Data.rAcc, 
                                    Dec         := Data.rDec, 
                                    Jerk        := Data.rJerk, 
                                    Direction   := Data.iDirection, 
                                    BufferMode  := Tc2_MC2.MC_BufferMode.MC_Aborting);
    IF (_eres = E_PROGRESS.ERROR)
    THEN
        _eState             := E_PROGRESS.ERROR;
    ELSIF (_eres = E_PROGRESS.DONE)
    THEN 
      _eState               := E_PROGRESS.WORKING;
    END_IF
END_CASE
CASE _eState
OF
  E_PROGRESS.WORKING:
    _eState                 := E_PROGRESS.DONE;
    _eres                   := MoveVelo(
                                    Execute     := FALSE, 
                                    Velocity    := Data.rSetVelo, 
                                    Acc         := Data.rAcc, 
                                    Dec         := Data.rDec, 
                                    Jerk        := Data.rJerk, 
                                    Direction   := Data.iDirection, 
                                    BufferMode  := Tc2_MC2.MC_BufferMode.MC_Aborting);

END_CASE

MoveVelocity := _eState;
END_METHOD

PROPERTY MultiMasterGearIn : pointer to ARRAY[1..PLC_CONSTANT.MAX_AXIS] OF ST_GEAR_IN
SET
_GearMultiMasterParameter := MultiMasterGearIn;
END_SET
END_PROPERTY

METHOD ParameterRead : E_PROGRESS
VAR_INPUT
  Execute           : BOOL;
  ParameterNr       : Tc2_MC2.MC_AxisParameter;
END_VAR
VAR_INST
  _eres,
  _eState           : E_PROGRESS;
  _rValue           : LREAL;
  _stMsg            : ST_Message;
END_VAR
IF NOT Check() THEN _eState := E_PROGRESS.ERROR; END_IF
IF NOT Execute THEN _eState := E_PROGRESS.INIT; END_IF

CASE _eState
OF
  E_PROGRESS.INIT:
    IF Execute 
    THEN
      memset(ADR(_stMsg),0,SIZEOF(_stMsg));
      _rValue                       := 0;
      _eState                       := E_PROGRESS.BUSY;
    END_IF
END_CASE
CASE _eState
OF
  E_PROGRESS.BUSY:
    _eState         := E_PROGRESS.WAITING;
    _eres           := ReadParameter(
                                  Execute         := FALSE,
                                  ParameterNumber := ParameterNr);
END_CASE
CASE _eState
OF
  E_PROGRESS.WAITING:
    _eres           := ReadParameter(
                                  Execute         := TRUE,
                                  ParameterNumber := ParameterNr);

    IF (_eres = E_PROGRESS.ERROR)
    THEN
        _eState     := E_PROGRESS.ERROR;
    ELSIF (_eres = E_PROGRESS.DONE)
    THEN 
      _eState       := E_PROGRESS.WORKING;
    END_IF

  E_PROGRESS.WORKING:
    _eres           := ReadParameter(
                                  Execute         := FALSE,
                                  ParameterNumber := ParameterNr);

    _NcParameter^[_nAxisIndex].rValue :=
    _rParameterReadValue              := ReadParameterValue;
    _eState                           := E_PROGRESS.DONE;
END_CASE

ParameterRead := _eState;
END_METHOD

METHOD ParameterWrite : E_PROGRESS
VAR_INPUT
  Execute           : BOOL;
  ParameterNr       : Tc2_MC2.MC_AxisParameter;
END_VAR
VAR_INST
  _eres,
  _eState           : E_PROGRESS;
  _rValue           : LREAL;
  _stMsg            : ST_Message;
END_VAR
IF NOT Check() THEN _eState := E_PROGRESS.ERROR; END_IF
IF NOT Execute THEN _eState := E_PROGRESS.INIT; END_IF

CASE _eState
OF
  E_PROGRESS.INIT:
    IF Execute 
    THEN
      memset(ADR(_stMsg),0,SIZEOF(_stMsg));
      _rValue                     := _NcParameter^[_nAxisIndex].rValue;
      _eState                     := E_PROGRESS.BUSY;
    END_IF
END_CASE
CASE _eState
OF
  E_PROGRESS.BUSY:
    _eState         := E_PROGRESS.WAITING;
    _eres           := WriteParameter(
                                  Execute         := FALSE,
                                  Value           := _rValue,
                                  ParameterNumber := ParameterNr);
END_CASE
CASE _eState
OF
  E_PROGRESS.WAITING:
    _eres           := WriteParameter(
                                  Execute         := TRUE,
                                  Value           := _rValue,
                                  ParameterNumber := ParameterNr);

    IF (_eres = E_PROGRESS.ERROR)
    THEN
        _eState     := E_PROGRESS.ERROR;
    ELSIF (_eres = E_PROGRESS.DONE)
    THEN 
      _eState       := E_PROGRESS.WORKING;
    END_IF

  E_PROGRESS.WORKING:
    _eres           := WriteParameter(
                                  Execute         := FALSE,
                                  Value           := _rValue,
                                  ParameterNumber := ParameterNr);

    _eState                       := E_PROGRESS.DONE;
END_CASE

ParameterWrite                    := _eState;
END_METHOD

METHOD ParameterWritePersistent : E_PROGRESS
VAR_INPUT
  Execute           : BOOL;
  ParameterNr       : Tc2_MC2.MC_AxisParameter;
END_VAR
VAR_INST
  _eres,
  _eState           : E_PROGRESS;
  _rValue           : LREAL;
  _stMsg            : ST_Message;
END_VAR
IF NOT Check() THEN _eState := E_PROGRESS.ERROR; END_IF
IF NOT Execute THEN _eState := E_PROGRESS.INIT; END_IF

CASE _eState
OF
  E_PROGRESS.INIT:
    IF Execute 
    THEN
      memset(ADR(_stMsg),0,SIZEOF(_stMsg));
      _rValue                     := _NcParameter^[_nAxisIndex].rValue;
      _eState                     := E_PROGRESS.BUSY;
    END_IF
END_CASE
CASE _eState
OF
  E_PROGRESS.BUSY:
    _eState         := E_PROGRESS.WAITING;
    _eres           := WriteParameterPersistent(
                                  Execute         := FALSE,
                                  Value           := _rValue,
                                  ParameterNumber := ParameterNr);
END_CASE
CASE _eState
OF
  E_PROGRESS.WAITING:
    _eres           := WriteParameterPersistent(
                                  Execute         := TRUE,
                                  Value           := _rValue,
                                  ParameterNumber := ParameterNr);

    IF (_eres = E_PROGRESS.ERROR)
    THEN
        _eState     := E_PROGRESS.ERROR;
    ELSIF (_eres = E_PROGRESS.DONE)
    THEN 
      _eState       := E_PROGRESS.WORKING;
    END_IF

  E_PROGRESS.WORKING:
    _eres           := WriteParameterPersistent(
                                  Execute         := FALSE,
                                  Value           := _rValue,
                                  ParameterNumber := ParameterNr);

    _eState                       := E_PROGRESS.DONE;
END_CASE

ParameterWritePersistent          := _eState;
END_METHOD

METHOD PRIVATE ResetSoE : E_PROGRESS
VAR_INPUT
  Execute           : BOOL;
END_VAR
VAR_INST
  _eState           : E_PROGRESS;
  _rValue           : LREAL;
  _udiErrSer,
  _udiErrAds        : UDINT;
  _stMsg            : ST_Message;

	_fbReset		      : Tc2_MC2_Drive.FB_SoEReset;
  _tonDelay         : Tc2_Standard.TON;
	_nRepeat			    : UINT;

  _sErrorSercos     : Tc2_System.T_MaxString;

END_VAR
IF NOT Check() THEN _eState := E_PROGRESS.ERROR; END_IF
IF NOT Execute THEN _eState := E_PROGRESS.INIT; END_IF

CASE _eState
OF
  E_PROGRESS.INIT:
    IF Execute 
    THEN
      memset(ADR(_stMsg),0,SIZEOF(_stMsg));
      memset(ADR(_sErrorSercos),0,SIZEOF(_sErrorSercos));

		  _nRepeat                      := 1;
      _udiErrSer := _udiErrAds      := 0;
      _rValue                       := 0;
      _eState                       := E_PROGRESS.BUSY;
    END_IF
END_CASE
CASE _eState
OF
  E_PROGRESS.BUSY:
    _eState                         := E_PROGRESS.WAITING;
		_tonDelay(
            IN                      := FALSE);

		_fbReset(
            Execute                 := FALSE, 
            Timeout                 := T#2500MS, 
            Axis                    := _AxisRef^);
END_CASE
CASE _eState
OF
  E_PROGRESS.WAITING:
		_tonDelay(
            PT                      := T#1500MS, 
            IN                      := TRUE);

		_fbReset(
            Execute                 := TRUE, 
            Axis                    := _AxisRef^, 
            AdsErrId                => _udiErrAds, 
            SercosErrId             => _udiErrSer);

    IF _fbReset.Error
    THEN
      _stMsg.eType                  := E_MessageType.eMessageError;
      _stMsg.eDevice                := e_Device.Axis + TO_DINT(_AxisRef^.NcToPlc.AxisId);
      _stMsg.eSubdevice             :=  e_SubDevice.fbResetSercos;
      _stMsg.iErrorNumber           := _udiErrAds;

      _sErrorSercos                 := Tc2_Utilities.DATA_TO_HEXSTR(ADR(_udiErrSer), SIZEOF(_udiErrSer), FALSE);

      _stMsg.sText                  := concat('Sercos Err Nr: ', _sErrorSercos);

      f_MessageSet(_stMsg);

      _Info^[_nAxisIndex].nErrorId := _udiErrSer;
      _eState                       := E_PROGRESS.ERROR;

		ELSIF NOT _fbReset.Busy
		THEN
      _eState                       := E_PROGRESS.WORKING;

    ELSE
      IF _tonDelay.Q AND
         _AxisRef^.NcToPlc.StateDWord.28
      THEN
        _nRepeat                    := _nRepeat + 1;
        _eState                     := E_PROGRESS.BUSY;    
      END_IF

      IF (_nRepeat > 5)
      THEN
        _eState                     := E_PROGRESS.ERROR;
      END_IF
		END_IF
END_CASE
CASE _eState
OF
  E_PROGRESS.WORKING:
    _eState                         := E_PROGRESS.DONE;
END_CASE


ResetSoE := _eState;
END_METHOD

PROPERTY TargetWindow : lreal
GET
END_GET
SET
END_SET
END_PROPERTY

METHOD Template : E_PROGRESS
VAR_INPUT
  Execute           : BOOL;
END_VAR
VAR_INST
  _eState           : E_PROGRESS;
  _rValue           : LREAL;
  _udiErr           : UDINT;
  _stMsg            : ST_Message;


END_VAR
IF NOT Check() THEN _eState := E_PROGRESS.ERROR; END_IF
IF NOT Execute THEN _eState := E_PROGRESS.INIT; END_IF

CASE _eState
OF
  E_PROGRESS.INIT:
    IF Execute 
    THEN
      memset(ADR(_stMsg),0,SIZEOF(_stMsg));
      _udiErr                       := 0;
      _rValue                       := 0;
      _eState                       := E_PROGRESS.BUSY;
    END_IF
END_CASE
CASE _eState
OF
  E_PROGRESS.BUSY:
    _eState                         := E_PROGRESS.STARTUP;
END_CASE
CASE _eState
OF
  E_PROGRESS.STARTUP:
    _eState                         := E_PROGRESS.PREPARE;
END_CASE
CASE _eState
OF
  E_PROGRESS.PREPARE:
    _eState                         := E_PROGRESS.READY;
END_CASE
CASE _eState
OF
  E_PROGRESS.READY:
    _eState                         := E_PROGRESS.WAITING;
END_CASE
CASE _eState
OF
  E_PROGRESS.WAITING:
    _eState                         := E_PROGRESS.WORKING;
END_CASE
CASE _eState
OF
  E_PROGRESS.WORKING:
    _eState                         := E_PROGRESS.DONE;
END_CASE

Template_1 := _eState;
END_METHOD

END_FUNCTION_BLOCK

(* stored: Version 1.1.0.1, ProductVersion 3.1.4024.12
   POU FB_AxisControl: Id {999335a0-5af6-0c1d-15bd-a65b83fb504c}, SpecialFunc None
   Folder private: Id {72055c1e-ae08-0707-1b82-aa6a286c994c}
   Folder properties: Id {ec33a634-95a7-05e3-1cf2-1ebdb2bd51b4}
   Property AxisCtrl: Id {6f4cd776-1490-073c-2411-2e9fa9e9a6b2}
   Set Set: Id {e630f942-2d4d-05b1-0f59-706c62e18b88}
   Property AxisData: Id {dd1871a7-f253-01d5-39fc-b8e8ee980c20}
   Set Set: Id {3a83fd26-6575-0237-0d2c-1c41a74f695f}
   Method AxisDisable: Id {5b07de5c-833d-0c24-00ad-ad559c3149a3}
   Method AxisEnable: Id {bdedff7a-4ac5-01d7-2a4e-56553b33f7f1}
   Property AxisGearInParameter: Id {b3665f5f-7d61-0534-18c3-fc4c139bfd64}
   Set Set: Id {c3054604-2569-09a1-2cae-8365cfdd1ede}
   Method AxisHalt: Id {9b3aecb2-f7be-0371-1558-f6e3e61aa21b}
   Method AxisHome: Id {4affed04-b463-0d9f-01c5-e55d9c21fdc1}
   Property AxisIndex: Id {ec26ef16-42cd-03a5-0740-028e92c264af}
   Set Set: Id {72c20e5d-c07d-04e2-2e7f-3065a8d113f1}
   Property AxisInfo: Id {43262739-6eeb-0240-259b-c24a2b7c9b8b}
   Set Set: Id {9f325ee6-0044-0408-1b8f-3ba89b0236ae}
   Method AxisInit: Id {cfb847c0-d387-0e90-3f6c-326032cd73b0}
   Property AxisNcParameter: Id {a00e8910-77c8-0a98-3ecf-242a3b2549b9}
   Set Set: Id {15199a8a-b1d7-019e-133f-411483cbf6d2}
   Property AxisNcParameterValue: Id {4f83dc68-3391-08cc-2ba6-0dca5b6f9170}
   Get Get: Id {c17f1740-3dbe-0323-21bb-d695e230a5f7}
   Method AxisReset: Id {983134b4-72eb-0c42-3ead-aaa67397970d}
   Property AxisState: Id {3dca1f6c-4c2d-0a02-0ad3-e24fa848690b}
   Set Set: Id {03f024e1-d54b-0d56-094a-cef330b0eb6d}
   Method AxisStop: Id {4a327d1b-00a7-09b1-2b27-f1512672b30e}
   Method Check: Id {f8c19456-13e2-0915-179c-dd36c10cb739}
   Method Cmd: Id {1389b619-e85f-0feb-358b-830cf714b972}
   Method GetCalibrationCam: Id {cce8967b-3b33-0d3c-2e17-bfaefcd5c5f7}
   Property HomingParameter: Id {bbed7ae6-3372-0209-2101-be3ac0cae96a}
   Set Set: Id {2a0c1316-16a0-0fe7-392a-ae61fe490c44}
   Method Idle: Id {91e094ba-3637-045f-257e-8b0236a82b6e}
   Method LogControl: Id {d80366c5-11f3-0a8a-297c-4979ebf61c8a}
   Method LogResult: Id {6a095a86-ad22-09b9-1058-5124e0b4c567}
   Property MotionOptions: Id {923ce8f8-17ae-0577-329b-a9bd138026ab}
   Set Set: Id {3c68ebc7-a095-0efe-0dd0-71092a4ee16d}
   Method MoveBufferPos: Id {8bea1fe6-78db-0d06-2903-94e698371421}
   Method MoveBufferVelo: Id {374fe133-fb4a-0fd3-3a5b-fe68bfd11804}
   Method MovePosition: Id {27760da5-88ba-02a4-20e2-a43d8fea6b68}
   Method MoveVelocity: Id {636baf69-d370-0962-3889-6678baa38f82}
   Property MultiMasterGearIn: Id {7a83f5f4-5ff0-0cd2-16a1-3b0e107b1074}
   Set Set: Id {88b1ac6e-2512-0af5-0f4b-f9a0ff532dc3}
   Method ParameterRead: Id {e888c5ae-12ad-0616-229c-9fc3342dcc87}
   Method ParameterWrite: Id {77ad02f2-e55b-0375-1054-18aeccc4f797}
   Method ParameterWritePersistent: Id {bfd2219d-61cd-01fc-2d61-aa05055375fb}
   Method ResetSoE: Id {4d30f9e6-607e-0983-163c-f478b48c7089}
   Property TargetWindow: Id {11d68468-93e3-0097-23b1-e0b3bcb90db4}
   Get Get: Id {0f08b6bc-07d3-0b4c-37b4-d89d0cb7c963}
   Set Set: Id {57184c7f-cacd-0caa-26dc-e19203ff97eb}
   Method Template: Id {f7a6377b-3c3c-04fd-3517-7f39ac13b38f} *)
